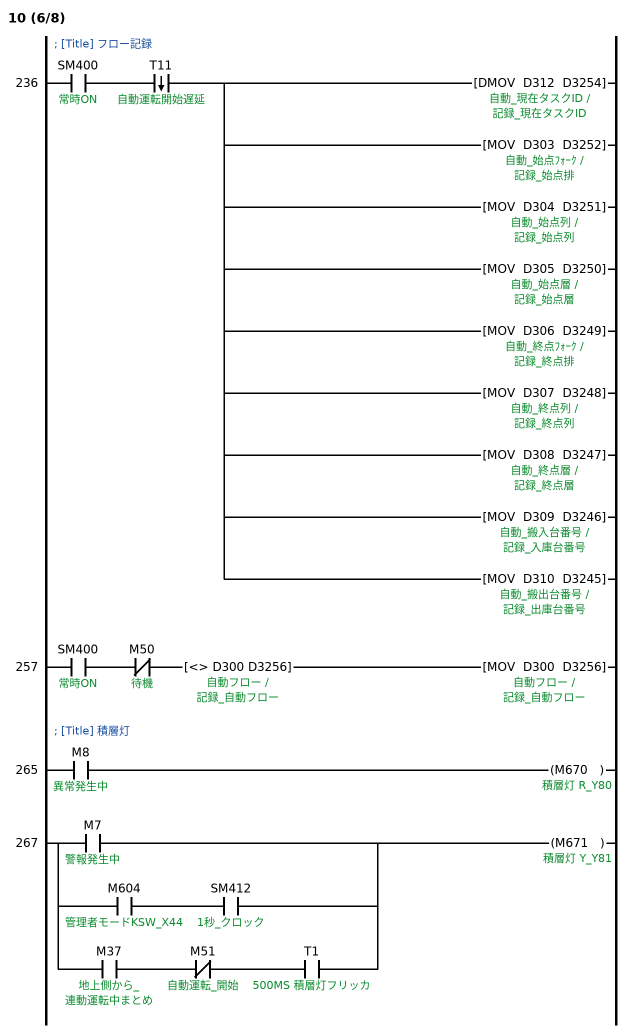
; [Title] フロー記録
236   LD      SM400  ; 常時ON
      ANDF    T11  ; 自動運転開始遅延
      DMOV    D312 D3254  ; 自動_現在タスクID / 記録_現在タスクID
      MOV     D303 D3252  ; 記録_始点排
      MOV     D304 D3251  ; 記録_始点列
      MOV     D305 D3250  ; 記録_始点層
      MOV     D306 D3249  ; 記録_終点排
      MOV     D307 D3248  ; 記録_終点列
      MOV     D308 D3247  ; 記録_終点層
      MOV     D309 D3246  ; 記録_入庫台番号
      MOV     D310 D3245  ; 記録_出庫台番号
257   LD      SM400  ; 常時ON
      ANI     M50  ; 待機
      AND<>   D300 D3256  ; 自動フロー / 記録_自動フロー
      MOV     D300 D3256
; [Title] 積層灯
265   LD      M8  ; 異常発生中
      OUT     M670  ; 積層灯 R_Y80
267   LD      M7  ; 警報発生中
      LD      M604  ; 管理者モードKSW_X44
      AND     SM412  ; 1秒_クロック
      ORB
      LD      M37  ; 地上側から_連動運転中まとめ
      ANI     M51  ; 自動運転_開始
      AND     T1  ; 500MS 積層灯フリッカ
      ORB
      OUT     M671  ; 積層灯 Y_Y81
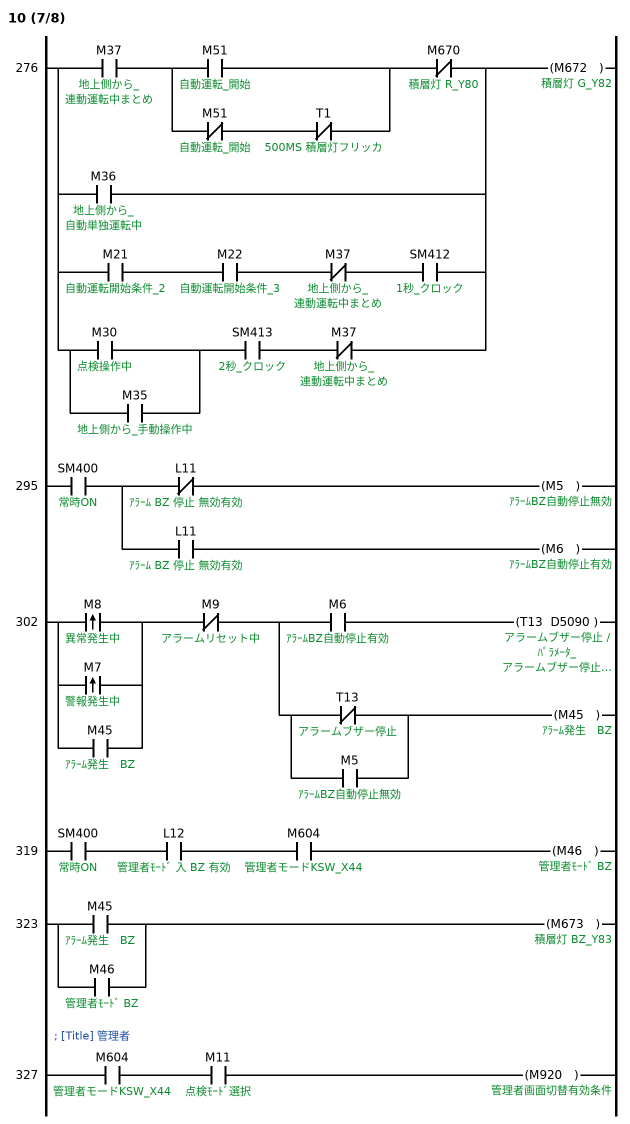
276   LD      M37  ; 地上側から_連動運転中まとめ
      LD      M51  ; 自動運転_開始
      LDI     M51  ; 自動運転_開始
      ANI     T1  ; 500MS 積層灯フリッカ
      ORB
      ANB
      ANI     M670  ; 積層灯 R_Y80
      OR      M36  ; 地上側から_自動単独運転中
      LD      M21  ; 自動運転開始条件_2
      AND     M22  ; 自動運転開始条件_3
      ANI     M37  ; 地上側から_連動運転中まとめ
      AND     SM412  ; 1秒_クロック
      ORB
      LD      M30  ; 点検操作中
      OR      M35  ; 地上側から_手動操作中
      AND     SM413  ; 2秒_クロック
      ANI     M37  ; 地上側から_連動運転中まとめ
      ORB
      OUT     M672  ; 積層灯 G_Y82
295   LD      SM400  ; 常時ON
      MPS
      ANI     L11  ; ｱﾗｰﾑ BZ 停止 無効有効
      OUT     M5  ; ｱﾗｰﾑBZ自動停止無効
      MPP
      AND     L11  ; ｱﾗｰﾑ BZ 停止 無効有効
      OUT     M6  ; ｱﾗｰﾑBZ自動停止有効
302   LDP     M8  ; 異常発生中
      ORP     M7  ; 警報発生中
      OR      M45  ; ｱﾗｰﾑ発生　BZ
      ANI     M9  ; アラームリセット中
      MPS
      AND     M6  ; ｱﾗｰﾑBZ自動停止有効
      OUT     T13 D5090  ; アラームブザー停止 / ﾊﾟﾗﾒｰﾀ_アラームブザー停止設定値
      MPP
      LDI     T13  ; アラームブザー停止
      OR      M5  ; ｱﾗｰﾑBZ自動停止無効
      ANB
      OUT     M45  ; ｱﾗｰﾑ発生　BZ
319   LD      SM400  ; 常時ON
      AND     L12  ; 管理者ﾓｰﾄﾞ 入 BZ 有効
      AND     M604  ; 管理者モードKSW_X44
      OUT     M46  ; 管理者ﾓｰﾄﾞ BZ
323   LD      M45  ; ｱﾗｰﾑ発生　BZ
      OR      M46  ; 管理者ﾓｰﾄﾞ BZ
      OUT     M673  ; 積層灯 BZ_Y83
; [Title] 管理者
327   LD      M604  ; 管理者モードKSW_X44
      AND     M11  ; 点検ﾓｰﾄﾞ選択
      OUT     M920  ; 管理者画面切替有効条件
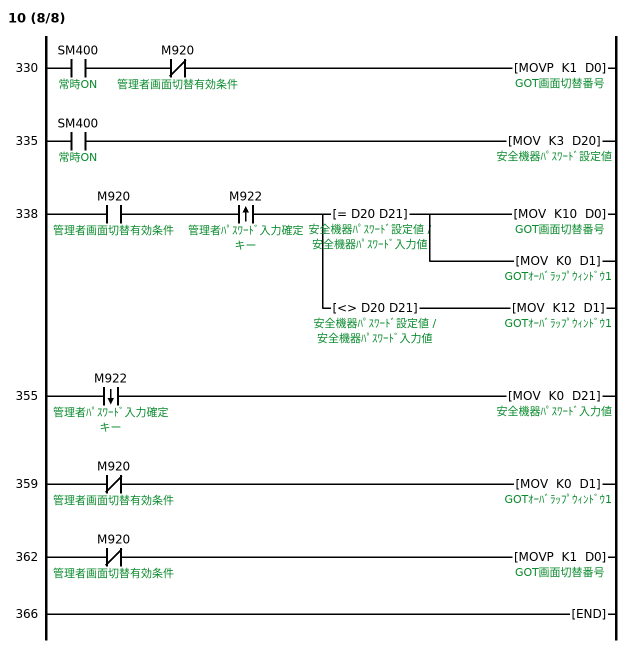
330   LD      SM400  ; 常時ON
      ANI     M920  ; 管理者画面切替有効条件
      MOVP    K1 D0  ; GOT画面切替番号
335   LD      SM400  ; 常時ON
      MOV     K3 D20  ; 安全機器ﾊﾟｽﾜｰﾄﾞ設定値
338   LD      M920  ; 管理者画面切替有効条件
      ANDP    M922  ; 管理者ﾊﾟｽﾜｰﾄﾞ入力確定キー
      MPS
      AND=    D20 D21  ; 安全機器ﾊﾟｽﾜｰﾄﾞ設定値 / 安全機器ﾊﾟｽﾜｰﾄﾞ入力値
      MOV     K10 D0
      MOV     K0 D1  ; GOTｵｰﾊﾞﾗｯﾌﾟｳｨﾝﾄﾞｳ1
      MPP
      AND<>   D20 D21  ; 安全機器ﾊﾟｽﾜｰﾄﾞ設定値 / 安全機器ﾊﾟｽﾜｰﾄﾞ入力値
      MOV     K12 D1
355   LDF     M922  ; 管理者ﾊﾟｽﾜｰﾄﾞ入力確定キー
      MOV     K0 D21
359   LDI     M920  ; 管理者画面切替有効条件
      MOV     K0 D1
362   LDI     M920  ; 管理者画面切替有効条件
      MOVP    K1 D0
366   END
END_PROGRAM

PROGRAM 12  // Stacker制御_自動
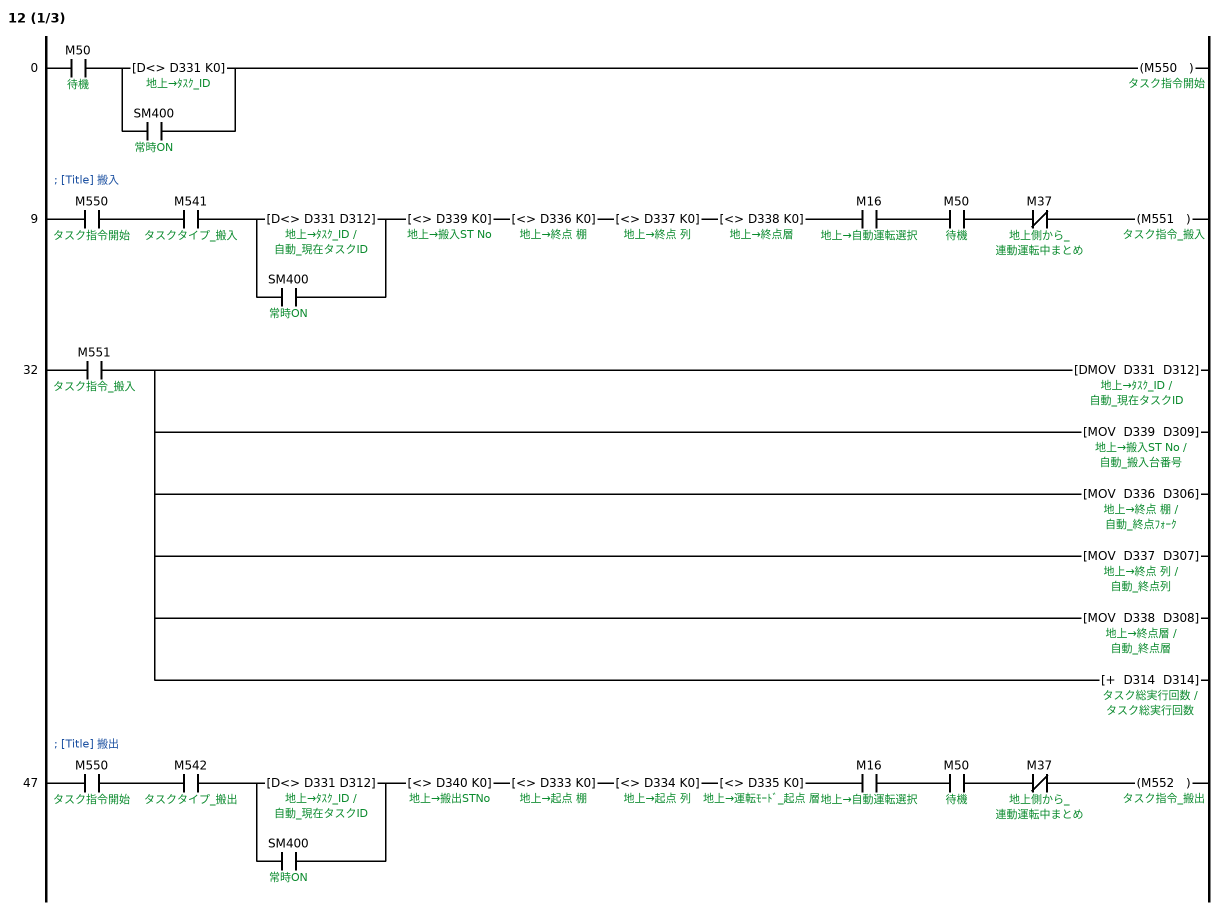
0     LD      M50  ; 待機
      LDD<>   D331 K0  ; 地上→ﾀｽｸ_ID
      OR      SM400  ; 常時ON
      ANB
      OUT     M550  ; タスク指令開始
; [Title] 搬入
9     LD      M550  ; タスク指令開始
      AND     M541  ; タスクタイプ_搬入
      LDD<>   D331 D312  ; 地上→ﾀｽｸ_ID / 自動_現在タスクID
      OR      SM400  ; 常時ON
      ANB
      AND<>   D339 K0  ; 地上→搬入ST No
      AND<>   D336 K0  ; 地上→終点 棚
      AND<>   D337 K0  ; 地上→終点 列
      AND<>   D338 K0  ; 地上→終点層
      AND     M16  ; 地上→自動運転選択
      AND     M50  ; 待機
      ANI     M37  ; 地上側から_連動運転中まとめ
      OUT     M551  ; タスク指令_搬入
32    LD      M551  ; タスク指令_搬入
      DMOV    D331 D312
      MOV     D339 D309  ; 自動_搬入台番号
      MOV     D336 D306  ; 自動_終点ﾌｫｰｸ
      MOV     D337 D307  ; 自動_終点列
      MOV     D338 D308  ; 自動_終点層
      +       D314 D314  ; タスク総実行回数
; [Title] 搬出
47    LD      M550  ; タスク指令開始
      AND     M542  ; タスクタイプ_搬出
      LDD<>   D331 D312  ; 地上→ﾀｽｸ_ID / 自動_現在タスクID
      OR      SM400  ; 常時ON
      ANB
      AND<>   D340 K0  ; 地上→搬出STNo
      AND<>   D333 K0  ; 地上→起点 棚
      AND<>   D334 K0  ; 地上→起点 列
      AND<>   D335 K0  ; 地上→運転ﾓｰﾄﾞ_起点 層
      AND     M16  ; 地上→自動運転選択
      AND     M50  ; 待機
      ANI     M37  ; 地上側から_連動運転中まとめ
      OUT     M552  ; タスク指令_搬出
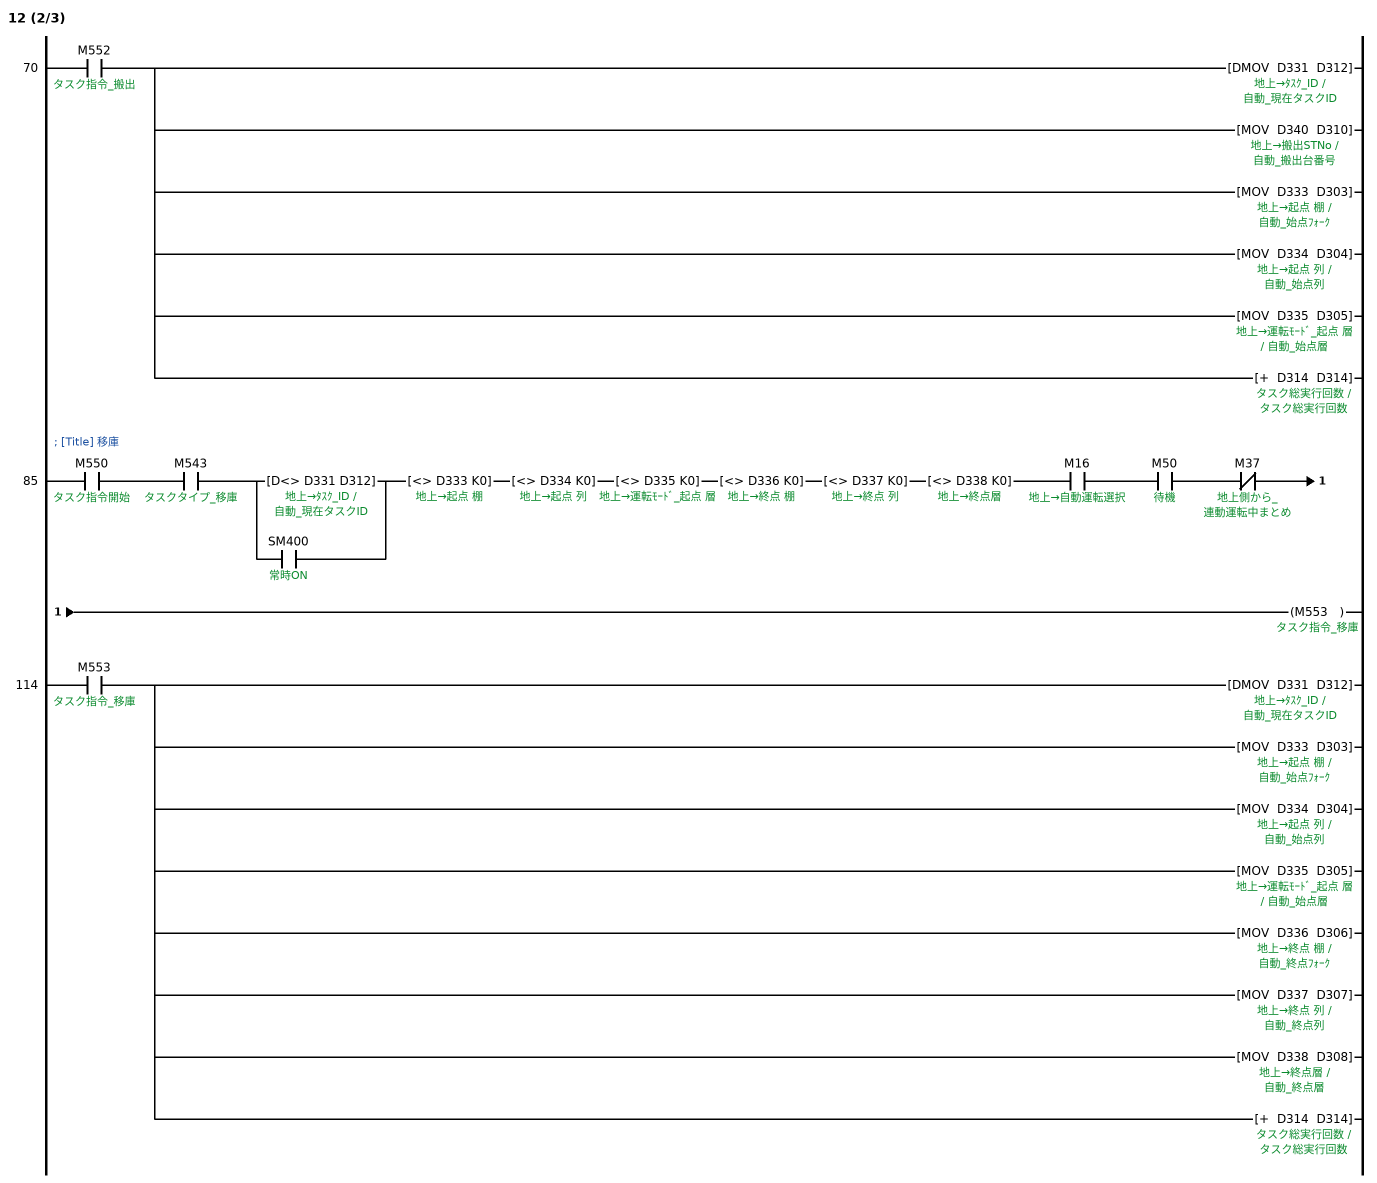
70    LD      M552  ; タスク指令_搬出
      DMOV    D331 D312
      MOV     D340 D310  ; 自動_搬出台番号
      MOV     D333 D303  ; 自動_始点ﾌｫｰｸ
      MOV     D334 D304  ; 自動_始点列
      MOV     D335 D305  ; 自動_始点層
      +       D314 D314
; [Title] 移庫
85    LD      M550  ; タスク指令開始
      AND     M543  ; タスクタイプ_移庫
      LDD<>   D331 D312  ; 地上→ﾀｽｸ_ID / 自動_現在タスクID
      OR      SM400  ; 常時ON
      ANB
      AND<>   D333 K0  ; 地上→起点 棚
      AND<>   D334 K0  ; 地上→起点 列
      AND<>   D335 K0  ; 地上→運転ﾓｰﾄﾞ_起点 層
      AND<>   D336 K0  ; 地上→終点 棚
      AND<>   D337 K0  ; 地上→終点 列
      AND<>   D338 K0  ; 地上→終点層
      AND     M16  ; 地上→自動運転選択
      AND     M50  ; 待機
      ANI     M37  ; 地上側から_連動運転中まとめ
      OUT     M553  ; タスク指令_移庫
114   LD      M553  ; タスク指令_移庫
      DMOV    D331 D312
      MOV     D333 D303
      MOV     D334 D304
      MOV     D335 D305
      MOV     D336 D306
      MOV     D337 D307
      MOV     D338 D308
      +       D314 D314
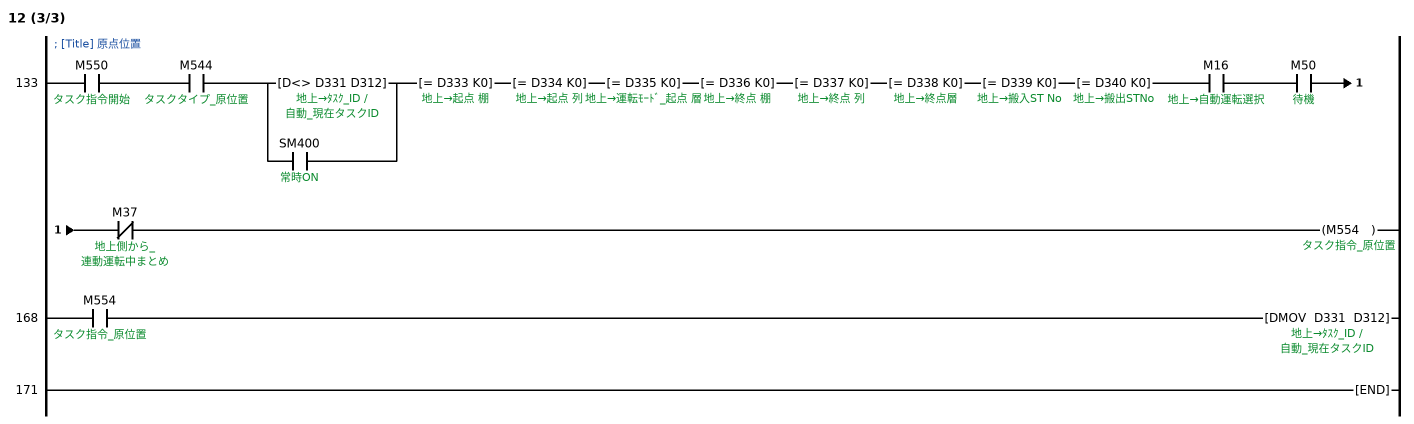
; [Title] 原点位置
133   LD      M550  ; タスク指令開始
      AND     M544  ; タスクタイプ_原位置
      LDD<>   D331 D312  ; 地上→ﾀｽｸ_ID / 自動_現在タスクID
      OR      SM400  ; 常時ON
      ANB
      AND=    D333 K0  ; 地上→起点 棚
      AND=    D334 K0  ; 地上→起点 列
      AND=    D335 K0  ; 地上→運転ﾓｰﾄﾞ_起点 層
      AND=    D336 K0  ; 地上→終点 棚
      AND=    D337 K0  ; 地上→終点 列
      AND=    D338 K0  ; 地上→終点層
      AND=    D339 K0  ; 地上→搬入ST No
      AND=    D340 K0  ; 地上→搬出STNo
      AND     M16  ; 地上→自動運転選択
      AND     M50  ; 待機
      ANI     M37  ; 地上側から_連動運転中まとめ
      OUT     M554  ; タスク指令_原位置
168   LD      M554  ; タスク指令_原位置
      DMOV    D331 D312
171   END
END_PROGRAM

PROGRAM 14  // 点検操作/地上側手動・自動単独
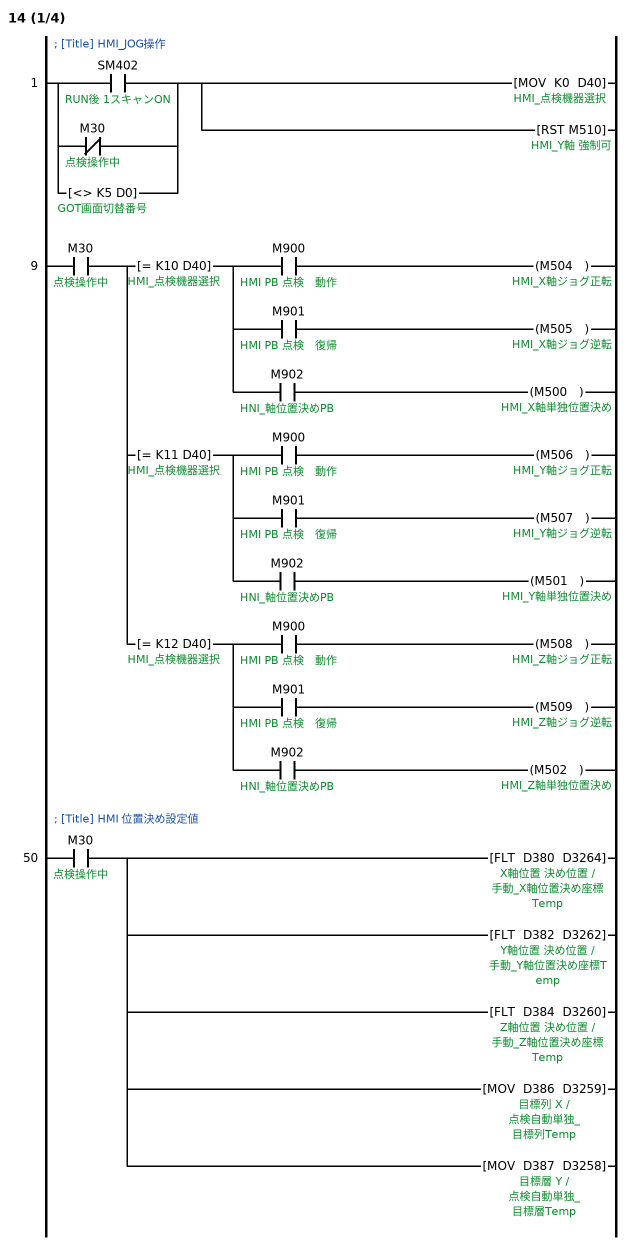
; [Title] HMI_JOG操作
1     LD      SM402  ; RUN後 1スキャンON
      ORI     M30  ; 点検操作中
      OR<>    K5 D0  ; GOT画面切替番号
      MOV     K0 D40  ; HMI_点検機器選択
      RST     M510  ; HMI_Y軸 強制可
9     LD      M30  ; 点検操作中
      MPS
      AND=    K10 D40  ; HMI_点検機器選択
      MPS
      AND     M900  ; HMI PB 点検　動作
      OUT     M504  ; HMI_X軸ジョグ正転
      MRD
      AND     M901  ; HMI PB 点検　復帰
      OUT     M505  ; HMI_X軸ジョグ逆転
      MPP
      AND     M902  ; HNI_軸位置決めPB
      OUT     M500  ; HMI_X軸単独位置決め
      MRD
      AND=    K11 D40  ; HMI_点検機器選択
      MPS
      AND     M900  ; HMI PB 点検　動作
      OUT     M506  ; HMI_Y軸ジョグ正転
      MRD
      AND     M901  ; HMI PB 点検　復帰
      OUT     M507  ; HMI_Y軸ジョグ逆転
      MPP
      AND     M902  ; HNI_軸位置決めPB
      OUT     M501  ; HMI_Y軸単独位置決め
      MPP
      AND=    K12 D40  ; HMI_点検機器選択
      MPS
      AND     M900  ; HMI PB 点検　動作
      OUT     M508  ; HMI_Z軸ジョグ正転
      MRD
      AND     M901  ; HMI PB 点検　復帰
      OUT     M509  ; HMI_Z軸ジョグ逆転
      MPP
      AND     M902  ; HNI_軸位置決めPB
      OUT     M502  ; HMI_Z軸単独位置決め
; [Title] HMI 位置決め設定値
50    LD      M30  ; 点検操作中
      FLT     D380 D3264  ; X軸位置 決め位置 / 手動_X軸位置決め座標Temp
      FLT     D382 D3262  ; Y軸位置 決め位置 / 手動_Y軸位置決め座標Temp
      FLT     D384 D3260  ; Z軸位置 決め位置 / 手動_Z軸位置決め座標Temp
      MOV     D386 D3259  ; 目標列 X / 点検自動単独_目標列Temp
      MOV     D387 D3258  ; 目標層 Y / 点検自動単独_目標層Temp
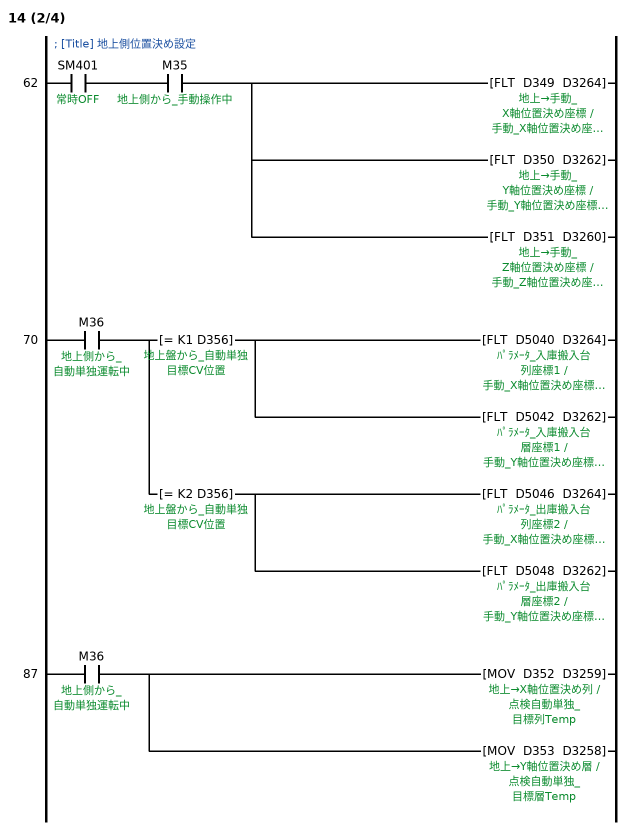
; [Title] 地上側位置決め設定
62    LD      SM401  ; 常時OFF
      AND     M35  ; 地上側から_手動操作中
      FLT     D349 D3264  ; 地上→手動_X軸位置決め座標
      FLT     D350 D3262  ; 地上→手動_Y軸位置決め座標
      FLT     D351 D3260  ; 地上→手動_Z軸位置決め座標
70    LD      M36  ; 地上側から_自動単独運転中
      MPS
      AND=    K1 D356  ; 地上盤から_自動単独 目標CV位置
      FLT     D5040 D3264  ; ﾊﾟﾗﾒｰﾀ_入庫搬入台  列座標1
      FLT     D5042 D3262  ; ﾊﾟﾗﾒｰﾀ_入庫搬入台  層座標1
      MPP
      AND=    K2 D356  ; 地上盤から_自動単独 目標CV位置
      FLT     D5046 D3264  ; ﾊﾟﾗﾒｰﾀ_出庫搬入台  列座標2
      FLT     D5048 D3262  ; ﾊﾟﾗﾒｰﾀ_出庫搬入台  層座標2
87    LD      M36  ; 地上側から_自動単独運転中
      MOV     D352 D3259  ; 地上→X軸位置決め列
      MOV     D353 D3258  ; 地上→Y軸位置決め層
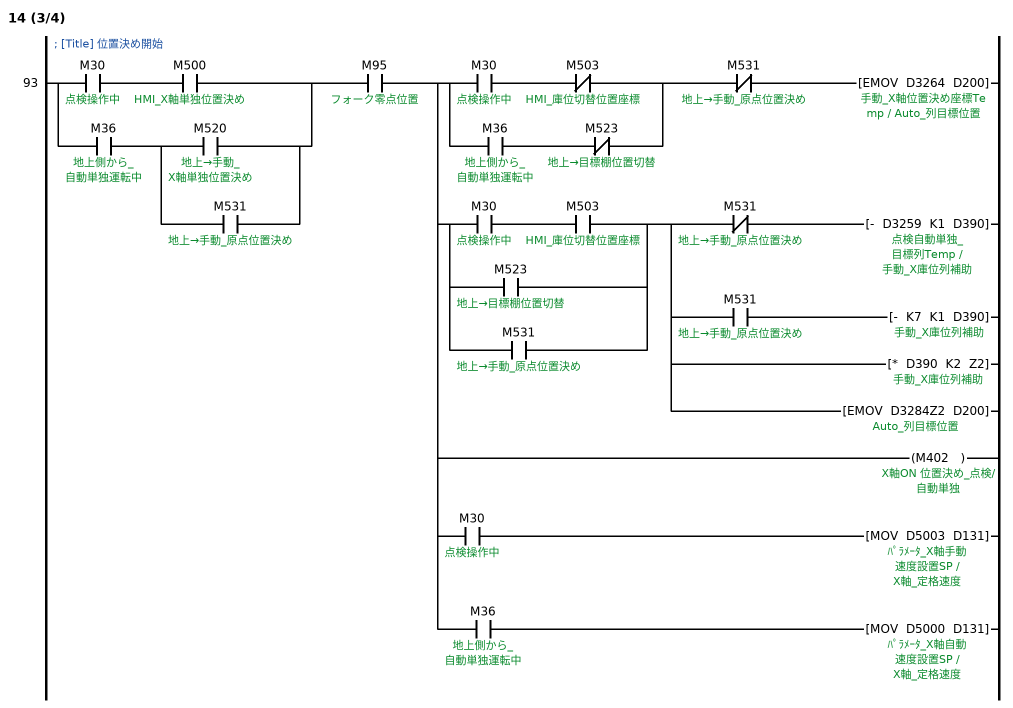
; [Title] 位置決め開始
93    LD      M30  ; 点検操作中
      AND     M500  ; HMI_X軸単独位置決め
      LD      M36  ; 地上側から_自動単独運転中
      LD      M520  ; 地上→手動_X軸単独位置決め
      OR      M531  ; 地上→手動_原点位置決め
      ANB
      ORB
      AND     M95  ; フォーク零点位置
      MPS
      LD      M30  ; 点検操作中
      ANI     M503  ; HMI_庫位切替位置座標
      LD      M36  ; 地上側から_自動単独運転中
      ANI     M523  ; 地上→目標棚位置切替
      ORB
      ANB
      ANI     M531  ; 地上→手動_原点位置決め
      EMOV    D3264 D200  ; Auto_列目標位置
      MRD
      LD      M30  ; 点検操作中
      AND     M503  ; HMI_庫位切替位置座標
      OR      M523  ; 地上→目標棚位置切替
      OR      M531  ; 地上→手動_原点位置決め
      ANB
      MPS
      ANI     M531  ; 地上→手動_原点位置決め
      -       D3259 K1 D390  ; 手動_X庫位列補助
      MRD
      AND     M531  ; 地上→手動_原点位置決め
      -       K7 K1 D390
      MPP
      *       D390 K2 Z2
      EMOV    D3284Z2 D200
      MPP
      OUT     M402  ; X軸ON 位置決め_点検/自動単独
      MPS
      AND     M30  ; 点検操作中
      MOV     D5003 D131  ; ﾊﾟﾗﾒｰﾀ_X軸手動 速度設置SP / X軸_定格速度
      MPP
      AND     M36  ; 地上側から_自動単独運転中
      MOV     D5000 D131  ; ﾊﾟﾗﾒｰﾀ_X軸自動 速度設置SP
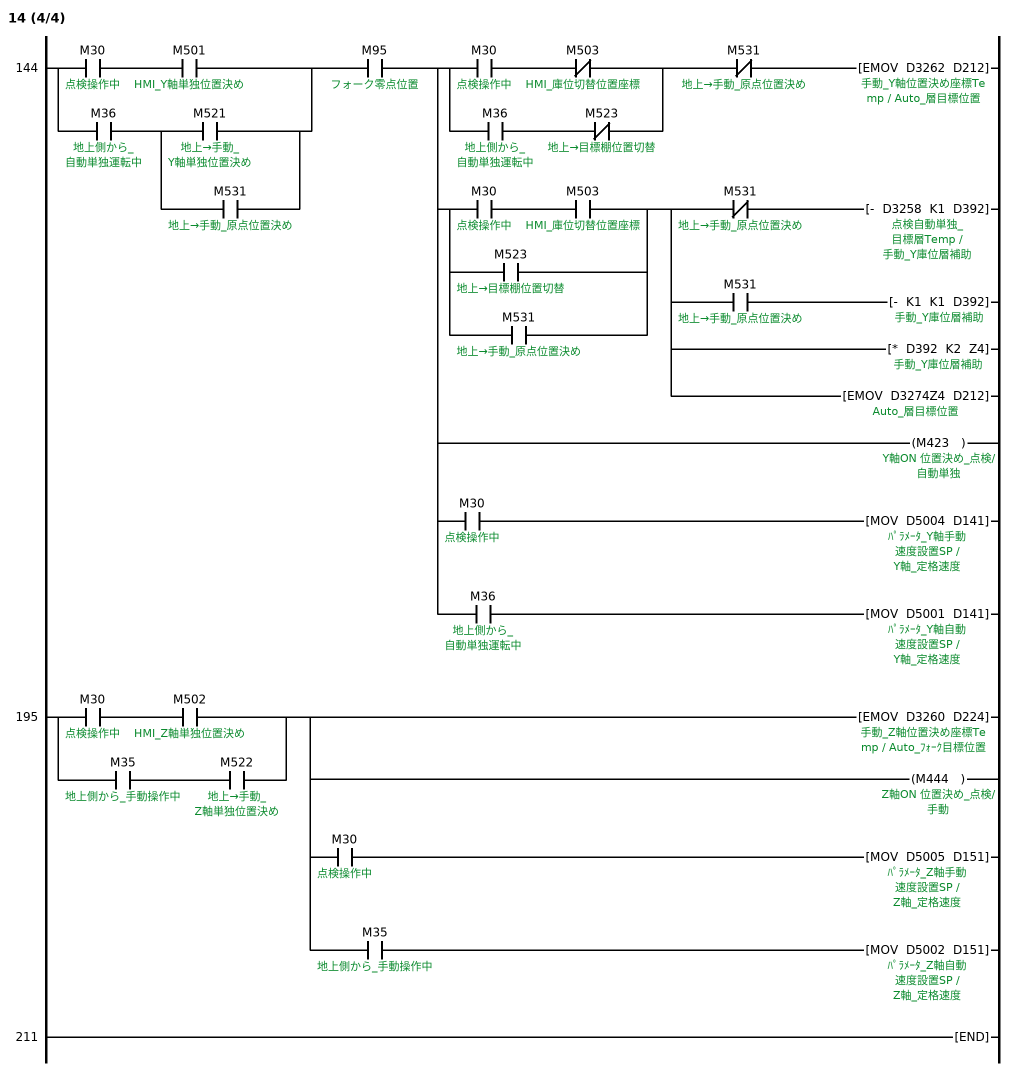
144   LD      M30  ; 点検操作中
      AND     M501  ; HMI_Y軸単独位置決め
      LD      M36  ; 地上側から_自動単独運転中
      LD      M521  ; 地上→手動_Y軸単独位置決め
      OR      M531  ; 地上→手動_原点位置決め
      ANB
      ORB
      AND     M95  ; フォーク零点位置
      MPS
      LD      M30  ; 点検操作中
      ANI     M503  ; HMI_庫位切替位置座標
      LD      M36  ; 地上側から_自動単独運転中
      ANI     M523  ; 地上→目標棚位置切替
      ORB
      ANB
      ANI     M531  ; 地上→手動_原点位置決め
      EMOV    D3262 D212  ; Auto_層目標位置
      MRD
      LD      M30  ; 点検操作中
      AND     M503  ; HMI_庫位切替位置座標
      OR      M523  ; 地上→目標棚位置切替
      OR      M531  ; 地上→手動_原点位置決め
      ANB
      MPS
      ANI     M531  ; 地上→手動_原点位置決め
      -       D3258 K1 D392  ; 手動_Y庫位層補助
      MRD
      AND     M531  ; 地上→手動_原点位置決め
      -       K1 K1 D392
      MPP
      *       D392 K2 Z4
      EMOV    D3274Z4 D212
      MPP
      OUT     M423  ; Y軸ON 位置決め_点検/自動単独
      MPS
      AND     M30  ; 点検操作中
      MOV     D5004 D141  ; ﾊﾟﾗﾒｰﾀ_Y軸手動 速度設置SP / Y軸_定格速度
      MPP
      AND     M36  ; 地上側から_自動単独運転中
      MOV     D5001 D141  ; ﾊﾟﾗﾒｰﾀ_Y軸自動 速度設置SP
195   LD      M30  ; 点検操作中
      AND     M502  ; HMI_Z軸単独位置決め
      LD      M35  ; 地上側から_手動操作中
      AND     M522  ; 地上→手動_Z軸単独位置決め
      ORB
      EMOV    D3260 D224  ; Auto_ﾌｫｰｸ目標位置
      OUT     M444  ; Z軸ON 位置決め_点検/手動
      MPS
      AND     M30  ; 点検操作中
      MOV     D5005 D151  ; ﾊﾟﾗﾒｰﾀ_Z軸手動 速度設置SP / Z軸_定格速度
      MPP
      AND     M35  ; 地上側から_手動操作中
      MOV     D5002 D151  ; ﾊﾟﾗﾒｰﾀ_Z軸自動 速度設置SP
211   END
END_PROGRAM

PROGRAM 15  // 軸制御
VAR
  AO1 : INT;
  __IST_24fe211bdc5e490f : I+ST_24fe211bdc5e490f;
  __IST_2ed1eb90aebe4c54 : I+ST_2ed1eb90aebe4c54;
  AO2 : INT;
END_VAR
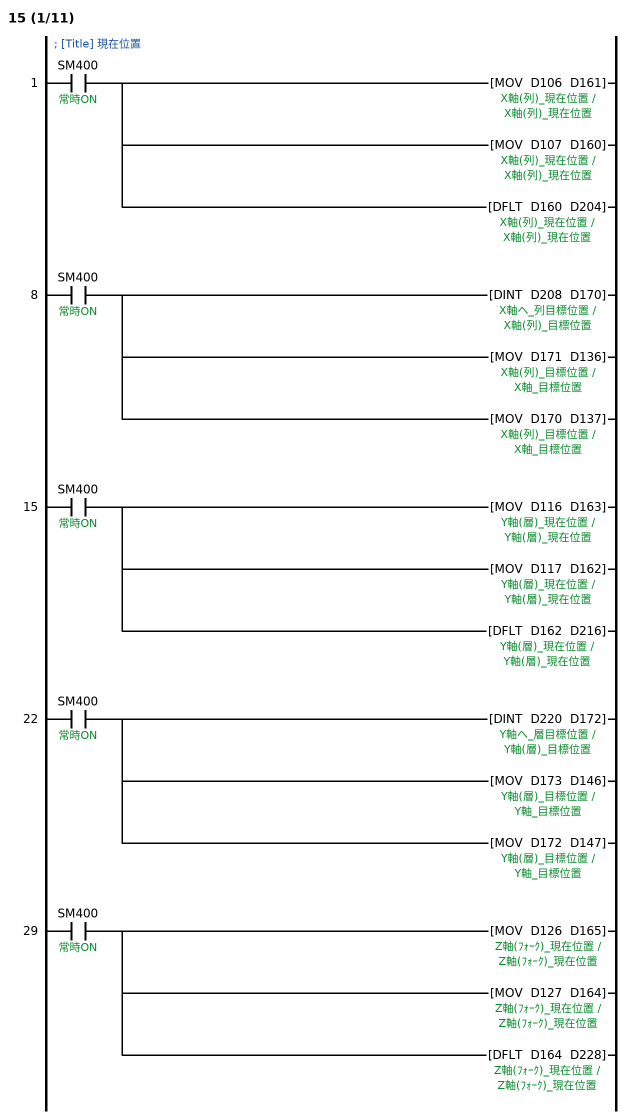
; [Title] 現在位置
1     LD      SM400  ; 常時ON
      MOV     D106 D161  ; X軸(列)_現在位置 / X軸(列)_現在位置
      MOV     D107 D160  ; X軸(列)_現在位置 / X軸(列)_現在位置
      DFLT    D160 D204  ; X軸(列)_現在位置
8     LD      SM400  ; 常時ON
      DINT    D208 D170  ; X軸へ_列目標位置 / X軸(列)_目標位置
      MOV     D171 D136  ; X軸(列)_目標位置 / X軸_目標位置
      MOV     D170 D137  ; X軸_目標位置
15    LD      SM400  ; 常時ON
      MOV     D116 D163  ; Y軸(層)_現在位置 / Y軸(層)_現在位置
      MOV     D117 D162  ; Y軸(層)_現在位置 / Y軸(層)_現在位置
      DFLT    D162 D216  ; Y軸(層)_現在位置
22    LD      SM400  ; 常時ON
      DINT    D220 D172  ; Y軸へ_層目標位置 / Y軸(層)_目標位置
      MOV     D173 D146  ; Y軸(層)_目標位置 / Y軸_目標位置
      MOV     D172 D147  ; Y軸_目標位置
29    LD      SM400  ; 常時ON
      MOV     D126 D165  ; Z軸(ﾌｫｰｸ)_現在位置 / Z軸(ﾌｫｰｸ)_現在位置
      MOV     D127 D164  ; Z軸(ﾌｫｰｸ)_現在位置 / Z軸(ﾌｫｰｸ)_現在位置
      DFLT    D164 D228  ; Z軸(ﾌｫｰｸ)_現在位置
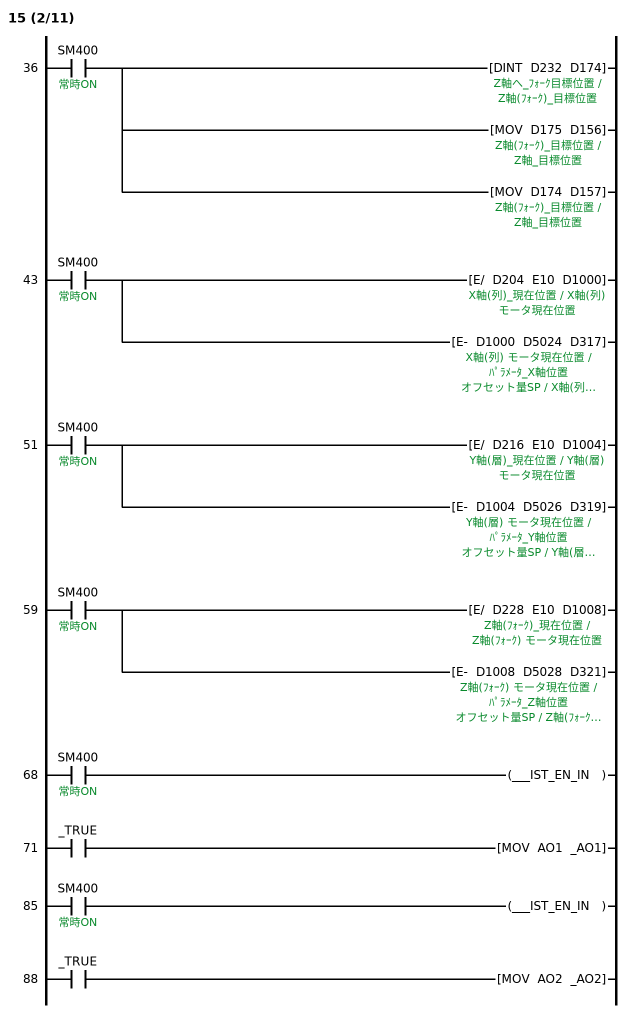
36    LD      SM400  ; 常時ON
      DINT    D232 D174  ; Z軸へ_ﾌｫｰｸ目標位置 / Z軸(ﾌｫｰｸ)_目標位置
      MOV     D175 D156  ; Z軸(ﾌｫｰｸ)_目標位置 / Z軸_目標位置
      MOV     D174 D157  ; Z軸_目標位置
43    LD      SM400  ; 常時ON
      E/      D204 E10 D1000  ; X軸(列) モータ現在位置
      E-      D1000 D5024 D317  ; ﾊﾟﾗﾒｰﾀ_X軸位置 オフセット量SP / X軸(列) 現在位置
51    LD      SM400  ; 常時ON
      E/      D216 E10 D1004  ; Y軸(層) モータ現在位置
      E-      D1004 D5026 D319  ; ﾊﾟﾗﾒｰﾀ_Y軸位置 オフセット量SP / Y軸(層) 現在位置
59    LD      SM400  ; 常時ON
      E/      D228 E10 D1008  ; Z軸(ﾌｫｰｸ) モータ現在位置
      E-      D1008 D5028 D321  ; ﾊﾟﾗﾒｰﾀ_Z軸位置 オフセット量SP / Z軸(ﾌｫｰｸ) 現在位置
; FB BLK START I+ST_24fe211bdc5e490f(__IST_24fe211bdc5e490f)
68    LD      SM400  ; 常時ON
      OUT     ___IST_EN_IN
71    LD      _TRUE
      MOV     AO1 _AO1
; FB START
; FB_NAME I+ST_24fe211bdc5e490f
; INSTANCE_NAME __IST_24fe211bdc5e490f
; FB IN_B:__IST_EN_IN
; FB OUT___IST_EN_OUT:B
; FB IN_W:AO1
; FB OUT_AO1:W
; FB END
; FB BLK END
; FB BLK START I+ST_2ed1eb90aebe4c54(__IST_2ed1eb90aebe4c54)
85    LD      SM400  ; 常時ON
      OUT     ___IST_EN_IN
88    LD      _TRUE
      MOV     AO2 _AO2
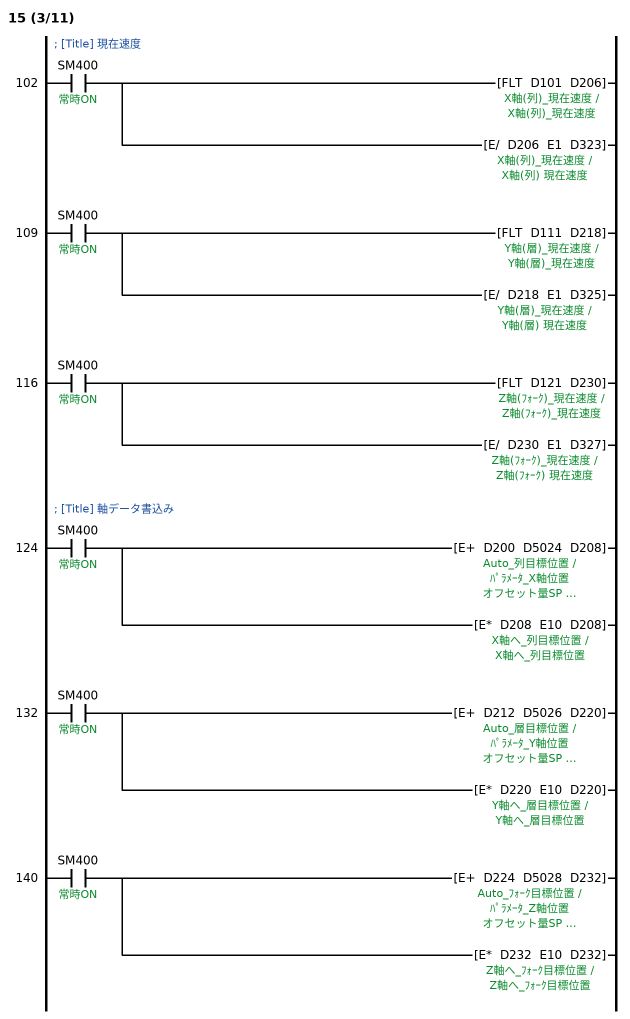
; FB START
; FB_NAME I+ST_2ed1eb90aebe4c54
; INSTANCE_NAME __IST_2ed1eb90aebe4c54
; FB IN_B:__IST_EN_IN
; FB OUT___IST_EN_OUT:B
; FB IN_W:AO2
; FB OUT_AO2:W
; FB END
; FB BLK END
; [Title] 現在速度
102   LD      SM400  ; 常時ON
      FLT     D101 D206  ; X軸(列)_現在速度 / X軸(列)_現在速度
      E/      D206 E1 D323  ; X軸(列) 現在速度
109   LD      SM400  ; 常時ON
      FLT     D111 D218  ; Y軸(層)_現在速度 / Y軸(層)_現在速度
      E/      D218 E1 D325  ; Y軸(層) 現在速度
116   LD      SM400  ; 常時ON
      FLT     D121 D230  ; Z軸(ﾌｫｰｸ)_現在速度 / Z軸(ﾌｫｰｸ)_現在速度
      E/      D230 E1 D327  ; Z軸(ﾌｫｰｸ) 現在速度
; [Title] 軸データ書込み
124   LD      SM400  ; 常時ON
      E+      D200 D5024 D208  ; Auto_列目標位置
      E*      D208 E10 D208
132   LD      SM400  ; 常時ON
      E+      D212 D5026 D220  ; Auto_層目標位置
      E*      D220 E10 D220
140   LD      SM400  ; 常時ON
      E+      D224 D5028 D232  ; Auto_ﾌｫｰｸ目標位置
      E*      D232 E10 D232
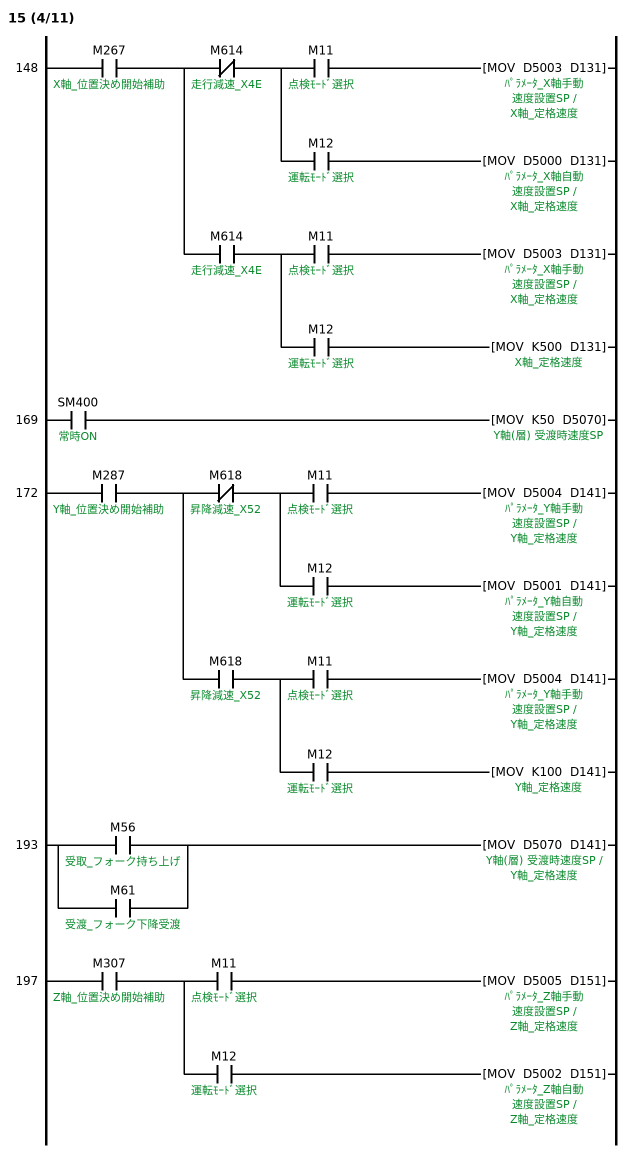
148   LD      M267  ; X軸_位置決め開始補助
      MPS
      ANI     M614  ; 走行減速_X4E
      MPS
      AND     M11  ; 点検ﾓｰﾄﾞ選択
      MOV     D5003 D131  ; ﾊﾟﾗﾒｰﾀ_X軸手動 速度設置SP / X軸_定格速度
      MPP
      AND     M12  ; 運転ﾓｰﾄﾞ選択
      MOV     D5000 D131  ; ﾊﾟﾗﾒｰﾀ_X軸自動 速度設置SP
      MPP
      AND     M614  ; 走行減速_X4E
      MPS
      AND     M11  ; 点検ﾓｰﾄﾞ選択
      MOV     D5003 D131
      MPP
      AND     M12  ; 運転ﾓｰﾄﾞ選択
      MOV     K500 D131
169   LD      SM400  ; 常時ON
      MOV     K50 D5070  ; Y軸(層) 受渡時速度SP
172   LD      M287  ; Y軸_位置決め開始補助
      MPS
      ANI     M618  ; 昇降減速_X52
      MPS
      AND     M11  ; 点検ﾓｰﾄﾞ選択
      MOV     D5004 D141  ; ﾊﾟﾗﾒｰﾀ_Y軸手動 速度設置SP / Y軸_定格速度
      MPP
      AND     M12  ; 運転ﾓｰﾄﾞ選択
      MOV     D5001 D141  ; ﾊﾟﾗﾒｰﾀ_Y軸自動 速度設置SP
      MPP
      AND     M618  ; 昇降減速_X52
      MPS
      AND     M11  ; 点検ﾓｰﾄﾞ選択
      MOV     D5004 D141
      MPP
      AND     M12  ; 運転ﾓｰﾄﾞ選択
      MOV     K100 D141
193   LD      M56  ; 受取_フォーク持ち上げ
      OR      M61  ; 受渡_フォーク下降受渡
      MOV     D5070 D141
197   LD      M307  ; Z軸_位置決め開始補助
      MPS
      AND     M11  ; 点検ﾓｰﾄﾞ選択
      MOV     D5005 D151  ; ﾊﾟﾗﾒｰﾀ_Z軸手動 速度設置SP / Z軸_定格速度
      MPP
      AND     M12  ; 運転ﾓｰﾄﾞ選択
      MOV     D5002 D151  ; ﾊﾟﾗﾒｰﾀ_Z軸自動 速度設置SP
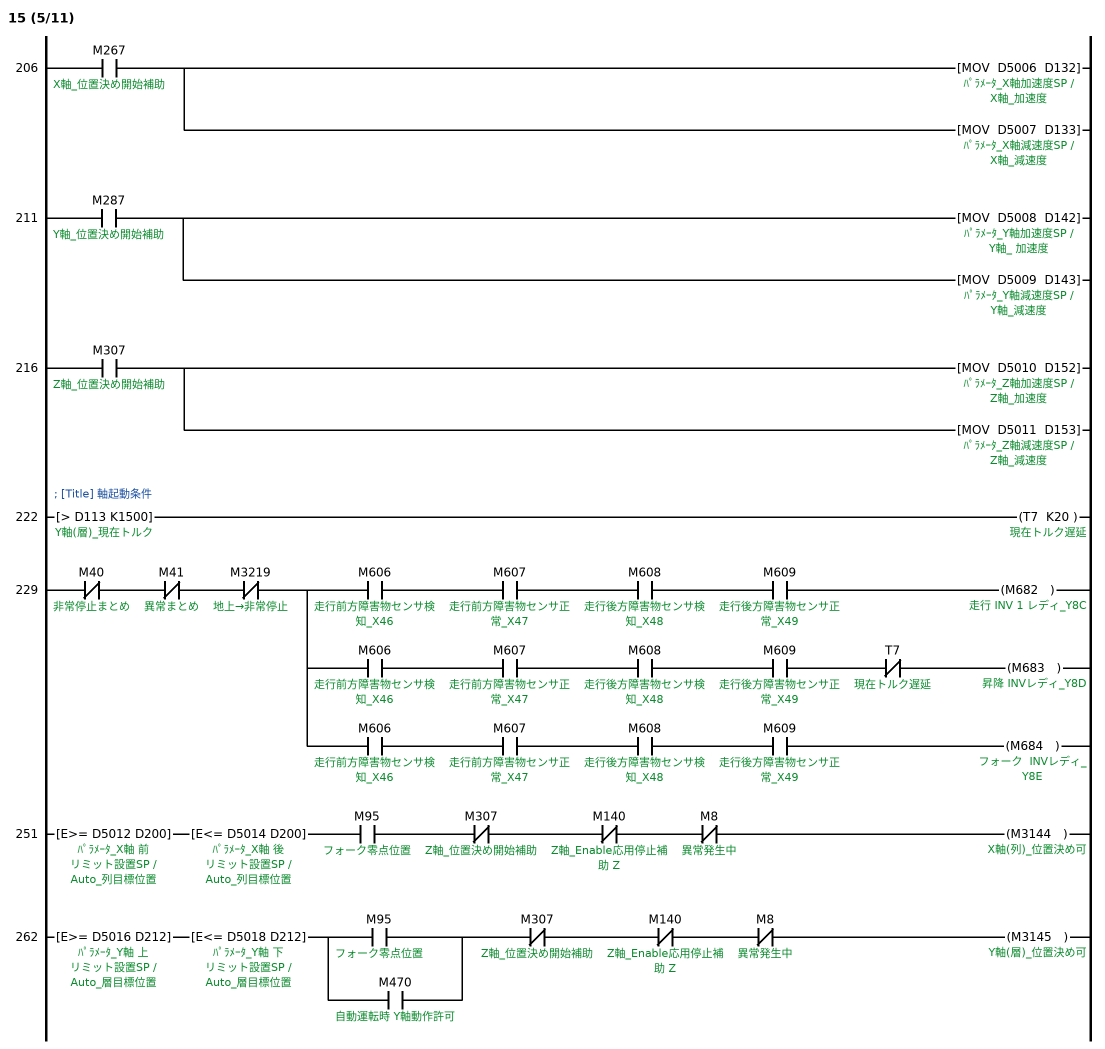
206   LD      M267  ; X軸_位置決め開始補助
      MOV     D5006 D132  ; ﾊﾟﾗﾒｰﾀ_X軸加速度SP / X軸_加速度
      MOV     D5007 D133  ; ﾊﾟﾗﾒｰﾀ_X軸減速度SP / X軸_減速度
211   LD      M287  ; Y軸_位置決め開始補助
      MOV     D5008 D142  ; ﾊﾟﾗﾒｰﾀ_Y軸加速度SP / Y軸_ 加速度
      MOV     D5009 D143  ; ﾊﾟﾗﾒｰﾀ_Y軸減速度SP / Y軸_減速度
216   LD      M307  ; Z軸_位置決め開始補助
      MOV     D5010 D152  ; ﾊﾟﾗﾒｰﾀ_Z軸加速度SP / Z軸_加速度
      MOV     D5011 D153  ; ﾊﾟﾗﾒｰﾀ_Z軸減速度SP / Z軸_減速度
; [Title] 軸起動条件
222   LD>     D113 K1500  ; Y軸(層)_現在トルク
      OUT     T7 K20  ; 現在トルク遅延
229   LDI     M40  ; 非常停止まとめ
      ANI     M41  ; 異常まとめ
      ANI     M3219  ; 地上→非常停止
      MPS
      AND     M606  ; 走行前方障害物センサ検知_X46
      AND     M607  ; 走行前方障害物センサ正常_X47
      AND     M608  ; 走行後方障害物センサ検知_X48
      AND     M609  ; 走行後方障害物センサ正常_X49
      OUT     M682  ; 走行 INV 1 レディ_Y8C
      MRD
      AND     M606  ; 走行前方障害物センサ検知_X46
      AND     M607  ; 走行前方障害物センサ正常_X47
      AND     M608  ; 走行後方障害物センサ検知_X48
      AND     M609  ; 走行後方障害物センサ正常_X49
      ANI     T7  ; 現在トルク遅延
      OUT     M683  ; 昇降 INVレディ_Y8D
      MPP
      AND     M606  ; 走行前方障害物センサ検知_X46
      AND     M607  ; 走行前方障害物センサ正常_X47
      AND     M608  ; 走行後方障害物センサ検知_X48
      AND     M609  ; 走行後方障害物センサ正常_X49
      OUT     M684  ; フォーク  INVレディ_Y8E
251   LDE>=   D5012 D200  ; ﾊﾟﾗﾒｰﾀ_X軸 前 リミット設置SP / Auto_列目標位置
      ANDE<=  D5014 D200  ; ﾊﾟﾗﾒｰﾀ_X軸 後 リミット設置SP / Auto_列目標位置
      AND     M95  ; フォーク零点位置
      ANI     M307  ; Z軸_位置決め開始補助
      ANI     M140  ; Z軸_Enable応用停止補助 Z
      ANI     M8  ; 異常発生中
      OUT     M3144  ; X軸(列)_位置決め可
262   LDE>=   D5016 D212  ; ﾊﾟﾗﾒｰﾀ_Y軸 上 リミット設置SP / Auto_層目標位置
      ANDE<=  D5018 D212  ; ﾊﾟﾗﾒｰﾀ_Y軸 下 リミット設置SP / Auto_層目標位置
      LD      M95  ; フォーク零点位置
      OR      M470  ; 自動運転時 Y軸動作許可
      ANB
      ANI     M307  ; Z軸_位置決め開始補助
      ANI     M140  ; Z軸_Enable応用停止補助 Z
      ANI     M8  ; 異常発生中
      OUT     M3145  ; Y軸(層)_位置決め可
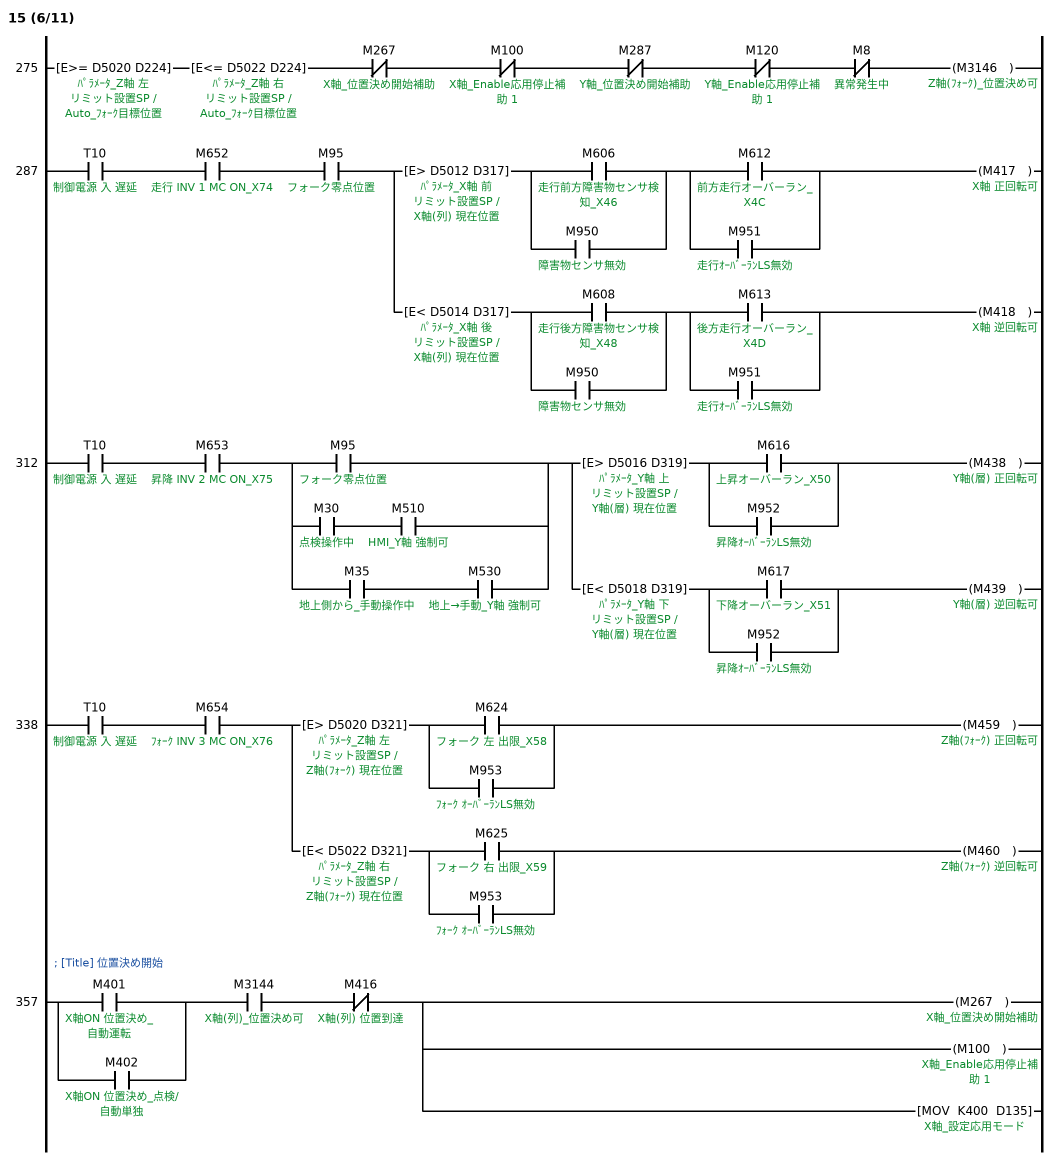
275   LDE>=   D5020 D224  ; ﾊﾟﾗﾒｰﾀ_Z軸 左 リミット設置SP / Auto_ﾌｫｰｸ目標位置
      ANDE<=  D5022 D224  ; ﾊﾟﾗﾒｰﾀ_Z軸 右 リミット設置SP / Auto_ﾌｫｰｸ目標位置
      ANI     M267  ; X軸_位置決め開始補助
      ANI     M100  ; X軸_Enable応用停止補助 1
      ANI     M287  ; Y軸_位置決め開始補助
      ANI     M120  ; Y軸_Enable応用停止補助 1
      ANI     M8  ; 異常発生中
      OUT     M3146  ; Z軸(ﾌｫｰｸ)_位置決め可
287   LD      T10  ; 制御電源 入 遅延
      AND     M652  ; 走行 INV 1 MC ON_X74
      AND     M95  ; フォーク零点位置
      MPS
      ANDE>   D5012 D317  ; ﾊﾟﾗﾒｰﾀ_X軸 前 リミット設置SP / X軸(列) 現在位置
      LD      M606  ; 走行前方障害物センサ検知_X46
      OR      M950  ; 障害物センサ無効
      ANB
      LD      M612  ; 前方走行オーバーラン_X4C
      OR      M951  ; 走行ｵｰﾊﾞｰﾗﾝLS無効
      ANB
      OUT     M417  ; X軸 正回転可
      MPP
      ANDE<   D5014 D317  ; ﾊﾟﾗﾒｰﾀ_X軸 後 リミット設置SP / X軸(列) 現在位置
      LD      M608  ; 走行後方障害物センサ検知_X48
      OR      M950  ; 障害物センサ無効
      ANB
      LD      M613  ; 後方走行オーバーラン_X4D
      OR      M951  ; 走行ｵｰﾊﾞｰﾗﾝLS無効
      ANB
      OUT     M418  ; X軸 逆回転可
312   LD      T10  ; 制御電源 入 遅延
      AND     M653  ; 昇降 INV 2 MC ON_X75
      LD      M95  ; フォーク零点位置
      LD      M30  ; 点検操作中
      AND     M510  ; HMI_Y軸 強制可
      ORB
      LD      M35  ; 地上側から_手動操作中
      AND     M530  ; 地上→手動_Y軸 強制可
      ORB
      ANB
      MPS
      ANDE>   D5016 D319  ; ﾊﾟﾗﾒｰﾀ_Y軸 上 リミット設置SP / Y軸(層) 現在位置
      LD      M616  ; 上昇オーバーラン_X50
      OR      M952  ; 昇降ｵｰﾊﾞｰﾗﾝLS無効
      ANB
      OUT     M438  ; Y軸(層) 正回転可
      MPP
      ANDE<   D5018 D319  ; ﾊﾟﾗﾒｰﾀ_Y軸 下 リミット設置SP / Y軸(層) 現在位置
      LD      M617  ; 下降オーバーラン_X51
      OR      M952  ; 昇降ｵｰﾊﾞｰﾗﾝLS無効
      ANB
      OUT     M439  ; Y軸(層) 逆回転可
338   LD      T10  ; 制御電源 入 遅延
      AND     M654  ; ﾌｫｰｸ INV 3 MC ON_X76
      MPS
      ANDE>   D5020 D321  ; ﾊﾟﾗﾒｰﾀ_Z軸 左 リミット設置SP / Z軸(ﾌｫｰｸ) 現在位置
      LD      M624  ; フォーク 左 出限_X58
      OR      M953  ; ﾌｫｰｸ ｵｰﾊﾞｰﾗﾝLS無効
      ANB
      OUT     M459  ; Z軸(ﾌｫｰｸ) 正回転可
      MPP
      ANDE<   D5022 D321  ; ﾊﾟﾗﾒｰﾀ_Z軸 右 リミット設置SP / Z軸(ﾌｫｰｸ) 現在位置
      LD      M625  ; フォーク 右 出限_X59
      OR      M953  ; ﾌｫｰｸ ｵｰﾊﾞｰﾗﾝLS無効
      ANB
      OUT     M460  ; Z軸(ﾌｫｰｸ) 逆回転可
; [Title] 位置決め開始
357   LD      M401  ; X軸ON 位置決め_自動運転
      OR      M402  ; X軸ON 位置決め_点検/自動単独
      AND     M3144  ; X軸(列)_位置決め可
      ANI     M416  ; X軸(列) 位置到達
      OUT     M267  ; X軸_位置決め開始補助
      OUT     M100  ; X軸_Enable応用停止補助 1
      MOV     K400 D135  ; X軸_設定応用モード
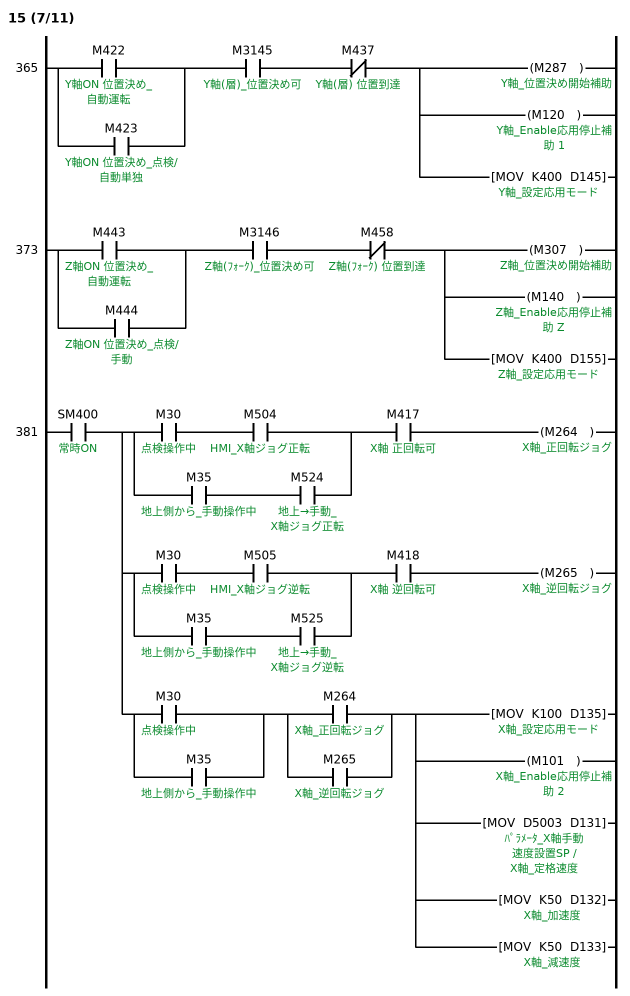
365   LD      M422  ; Y軸ON 位置決め_自動運転
      OR      M423  ; Y軸ON 位置決め_点検/自動単独
      AND     M3145  ; Y軸(層)_位置決め可
      ANI     M437  ; Y軸(層) 位置到達
      OUT     M287  ; Y軸_位置決め開始補助
      OUT     M120  ; Y軸_Enable応用停止補助 1
      MOV     K400 D145  ; Y軸_設定応用モード
373   LD      M443  ; Z軸ON 位置決め_自動運転
      OR      M444  ; Z軸ON 位置決め_点検/手動
      AND     M3146  ; Z軸(ﾌｫｰｸ)_位置決め可
      ANI     M458  ; Z軸(ﾌｫｰｸ) 位置到達
      OUT     M307  ; Z軸_位置決め開始補助
      OUT     M140  ; Z軸_Enable応用停止補助 Z
      MOV     K400 D155  ; Z軸_設定応用モード
381   LD      SM400  ; 常時ON
      MPS
      LD      M30  ; 点検操作中
      AND     M504  ; HMI_X軸ジョグ正転
      LD      M35  ; 地上側から_手動操作中
      AND     M524  ; 地上→手動_X軸ジョグ正転
      ORB
      ANB
      AND     M417  ; X軸 正回転可
      OUT     M264  ; X軸_正回転ジョグ
      MRD
      LD      M30  ; 点検操作中
      AND     M505  ; HMI_X軸ジョグ逆転
      LD      M35  ; 地上側から_手動操作中
      AND     M525  ; 地上→手動_X軸ジョグ逆転
      ORB
      ANB
      AND     M418  ; X軸 逆回転可
      OUT     M265  ; X軸_逆回転ジョグ
      MPP
      LD      M30  ; 点検操作中
      OR      M35  ; 地上側から_手動操作中
      ANB
      LD      M264  ; X軸_正回転ジョグ
      OR      M265  ; X軸_逆回転ジョグ
      ANB
      MOV     K100 D135
      OUT     M101  ; X軸_Enable応用停止補助 2
      MOV     D5003 D131
      MOV     K50 D132
      MOV     K50 D133
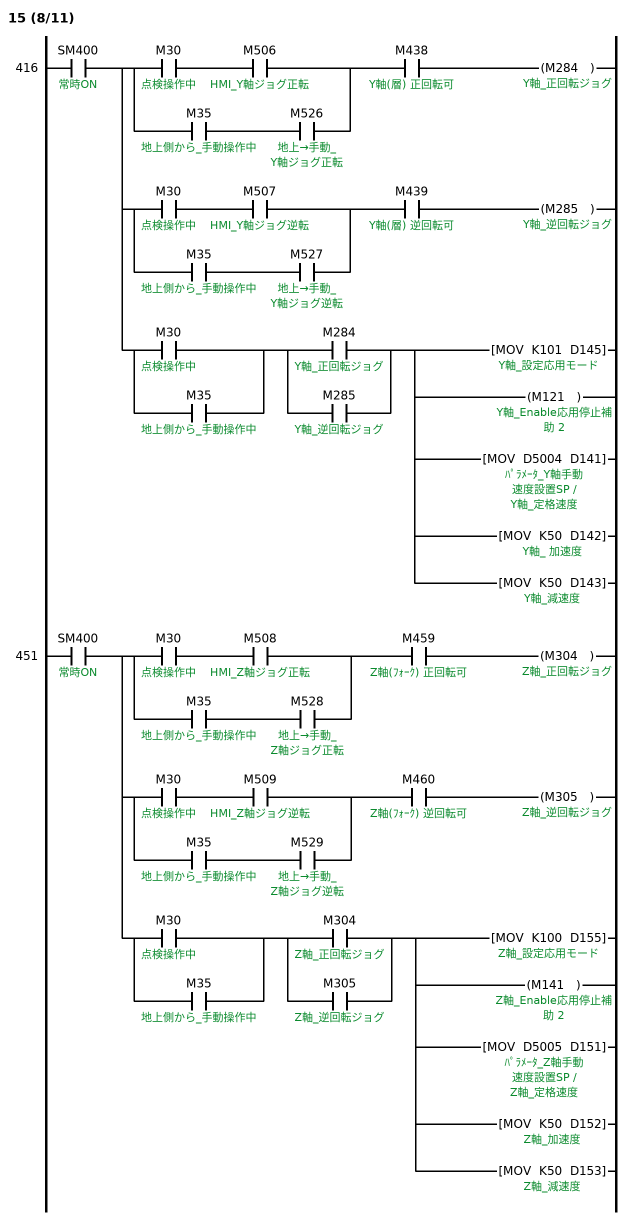
416   LD      SM400  ; 常時ON
      MPS
      LD      M30  ; 点検操作中
      AND     M506  ; HMI_Y軸ジョグ正転
      LD      M35  ; 地上側から_手動操作中
      AND     M526  ; 地上→手動_Y軸ジョグ正転
      ORB
      ANB
      AND     M438  ; Y軸(層) 正回転可
      OUT     M284  ; Y軸_正回転ジョグ
      MRD
      LD      M30  ; 点検操作中
      AND     M507  ; HMI_Y軸ジョグ逆転
      LD      M35  ; 地上側から_手動操作中
      AND     M527  ; 地上→手動_Y軸ジョグ逆転
      ORB
      ANB
      AND     M439  ; Y軸(層) 逆回転可
      OUT     M285  ; Y軸_逆回転ジョグ
      MPP
      LD      M30  ; 点検操作中
      OR      M35  ; 地上側から_手動操作中
      ANB
      LD      M284  ; Y軸_正回転ジョグ
      OR      M285  ; Y軸_逆回転ジョグ
      ANB
      MOV     K101 D145
      OUT     M121  ; Y軸_Enable応用停止補助 2
      MOV     D5004 D141
      MOV     K50 D142
      MOV     K50 D143
451   LD      SM400  ; 常時ON
      MPS
      LD      M30  ; 点検操作中
      AND     M508  ; HMI_Z軸ジョグ正転
      LD      M35  ; 地上側から_手動操作中
      AND     M528  ; 地上→手動_Z軸ジョグ正転
      ORB
      ANB
      AND     M459  ; Z軸(ﾌｫｰｸ) 正回転可
      OUT     M304  ; Z軸_正回転ジョグ
      MRD
      LD      M30  ; 点検操作中
      AND     M509  ; HMI_Z軸ジョグ逆転
      LD      M35  ; 地上側から_手動操作中
      AND     M529  ; 地上→手動_Z軸ジョグ逆転
      ORB
      ANB
      AND     M460  ; Z軸(ﾌｫｰｸ) 逆回転可
      OUT     M305  ; Z軸_逆回転ジョグ
      MPP
      LD      M30  ; 点検操作中
      OR      M35  ; 地上側から_手動操作中
      ANB
      LD      M304  ; Z軸_正回転ジョグ
      OR      M305  ; Z軸_逆回転ジョグ
      ANB
      MOV     K100 D155
      OUT     M141  ; Z軸_Enable応用停止補助 2
      MOV     D5005 D151
      MOV     K50 D152
      MOV     K50 D153
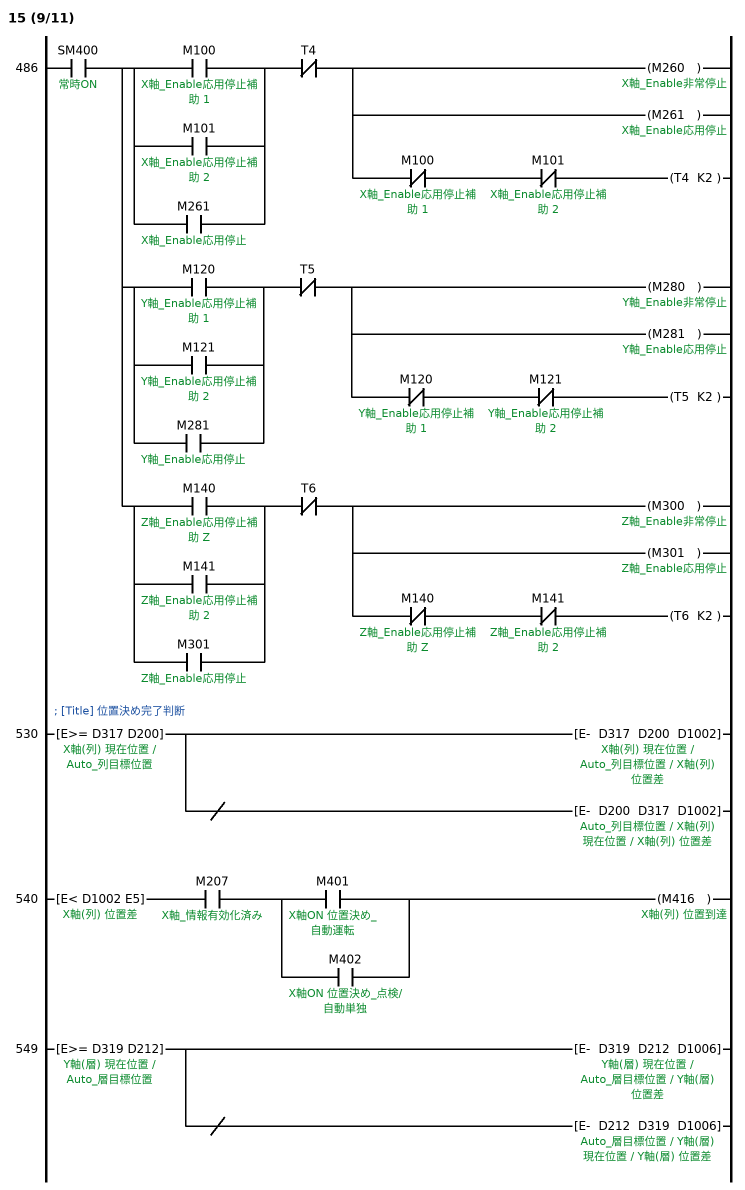
486   LD      SM400  ; 常時ON
      MPS
      LD      M100  ; X軸_Enable応用停止補助 1
      OR      M101  ; X軸_Enable応用停止補助 2
      OR      M261  ; X軸_Enable応用停止
      ANB
      ANI     T4
      OUT     M260  ; X軸_Enable非常停止
      OUT     M261  ; X軸_Enable応用停止
      ANI     M100  ; X軸_Enable応用停止補助 1
      ANI     M101  ; X軸_Enable応用停止補助 2
      OUT     T4 K2
      MRD
      LD      M120  ; Y軸_Enable応用停止補助 1
      OR      M121  ; Y軸_Enable応用停止補助 2
      OR      M281  ; Y軸_Enable応用停止
      ANB
      ANI     T5
      OUT     M280  ; Y軸_Enable非常停止
      OUT     M281  ; Y軸_Enable応用停止
      ANI     M120  ; Y軸_Enable応用停止補助 1
      ANI     M121  ; Y軸_Enable応用停止補助 2
      OUT     T5 K2
      MPP
      LD      M140  ; Z軸_Enable応用停止補助 Z
      OR      M141  ; Z軸_Enable応用停止補助 2
      OR      M301  ; Z軸_Enable応用停止
      ANB
      ANI     T6
      OUT     M300  ; Z軸_Enable非常停止
      OUT     M301  ; Z軸_Enable応用停止
      ANI     M140  ; Z軸_Enable応用停止補助 Z
      ANI     M141  ; Z軸_Enable応用停止補助 2
      OUT     T6 K2
; [Title] 位置決め完了判断
530   LDE>=   D317 D200  ; X軸(列) 現在位置 / Auto_列目標位置
      E-      D317 D200 D1002  ; X軸(列) 位置差
      INV
      E-      D200 D317 D1002
540   LDE<    D1002 E5  ; X軸(列) 位置差
      AND     M207  ; X軸_情報有効化済み
      LD      M401  ; X軸ON 位置決め_自動運転
      OR      M402  ; X軸ON 位置決め_点検/自動単独
      ANB
      OUT     M416  ; X軸(列) 位置到達
549   LDE>=   D319 D212  ; Y軸(層) 現在位置 / Auto_層目標位置
      E-      D319 D212 D1006  ; Y軸(層) 位置差
      INV
      E-      D212 D319 D1006
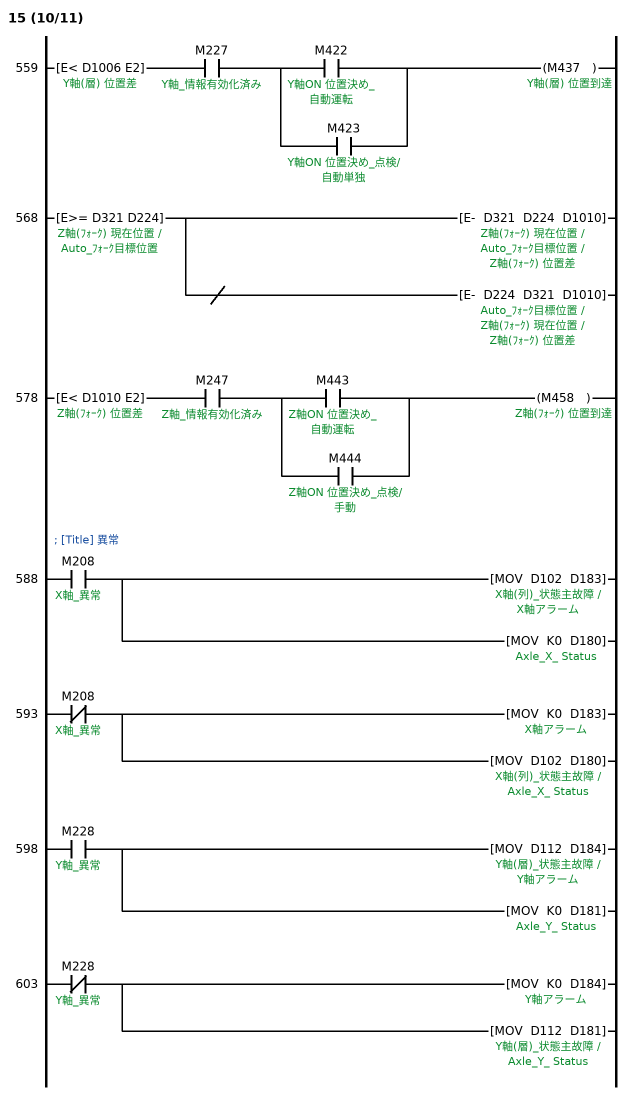
559   LDE<    D1006 E2  ; Y軸(層) 位置差
      AND     M227  ; Y軸_情報有効化済み
      LD      M422  ; Y軸ON 位置決め_自動運転
      OR      M423  ; Y軸ON 位置決め_点検/自動単独
      ANB
      OUT     M437  ; Y軸(層) 位置到達
568   LDE>=   D321 D224  ; Z軸(ﾌｫｰｸ) 現在位置 / Auto_ﾌｫｰｸ目標位置
      E-      D321 D224 D1010  ; Z軸(ﾌｫｰｸ) 位置差
      INV
      E-      D224 D321 D1010
578   LDE<    D1010 E2  ; Z軸(ﾌｫｰｸ) 位置差
      AND     M247  ; Z軸_情報有効化済み
      LD      M443  ; Z軸ON 位置決め_自動運転
      OR      M444  ; Z軸ON 位置決め_点検/手動
      ANB
      OUT     M458  ; Z軸(ﾌｫｰｸ) 位置到達
; [Title] 異常
588   LD      M208  ; X軸_異常
      MOV     D102 D183  ; X軸(列)_状態主故障 / X軸アラーム
      MOV     K0 D180  ; Axle_X_ Status
593   LDI     M208  ; X軸_異常
      MOV     K0 D183
      MOV     D102 D180
598   LD      M228  ; Y軸_異常
      MOV     D112 D184  ; Y軸(層)_状態主故障 / Y軸アラーム
      MOV     K0 D181  ; Axle_Y_ Status
603   LDI     M228  ; Y軸_異常
      MOV     K0 D184
      MOV     D112 D181
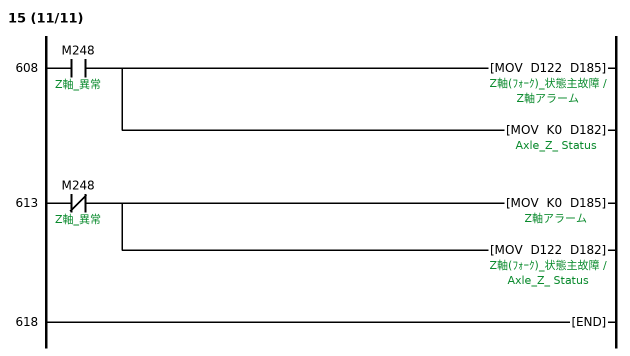
608   LD      M248  ; Z軸_異常
      MOV     D122 D185  ; Z軸(ﾌｫｰｸ)_状態主故障 / Z軸アラーム
      MOV     K0 D182  ; Axle_Z_ Status
613   LDI     M248  ; Z軸_異常
      MOV     K0 D185
      MOV     D122 D182
618   END
END_PROGRAM

PROGRAM 50  // I/O出力
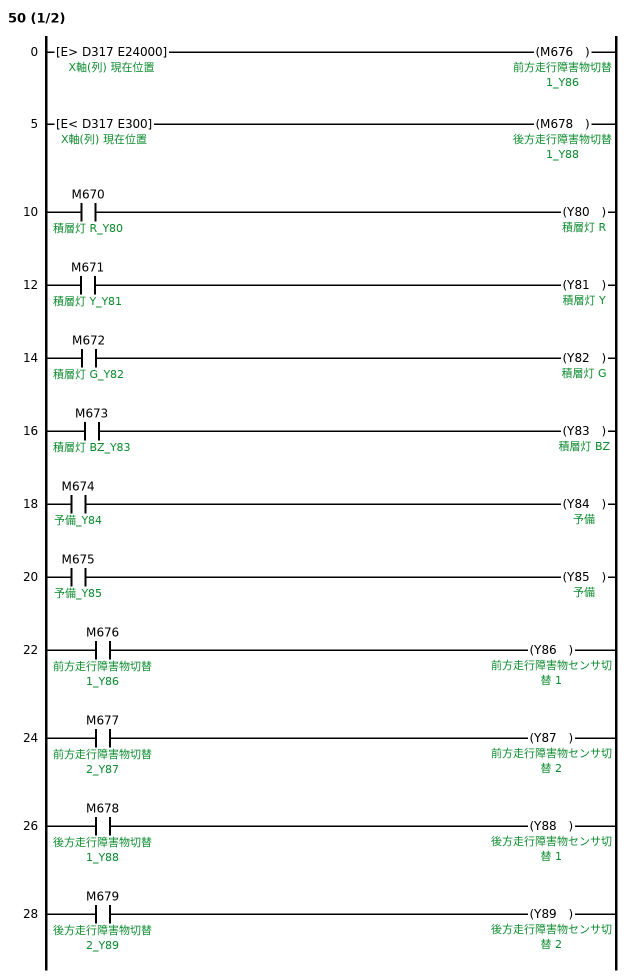
0     LDE>    D317 E24000  ; X軸(列) 現在位置
      OUT     M676  ; 前方走行障害物切替 1_Y86
5     LDE<    D317 E300  ; X軸(列) 現在位置
      OUT     M678  ; 後方走行障害物切替 1_Y88
10    LD      M670  ; 積層灯 R_Y80
      OUT     Y80  ; 積層灯 R
12    LD      M671  ; 積層灯 Y_Y81
      OUT     Y81  ; 積層灯 Y
14    LD      M672  ; 積層灯 G_Y82
      OUT     Y82  ; 積層灯 G
16    LD      M673  ; 積層灯 BZ_Y83
      OUT     Y83  ; 積層灯 BZ
18    LD      M674  ; 予備_Y84
      OUT     Y84  ; 予備
20    LD      M675  ; 予備_Y85
      OUT     Y85  ; 予備
22    LD      M676  ; 前方走行障害物切替 1_Y86
      OUT     Y86  ; 前方走行障害物センサ切替 1
24    LD      M677  ; 前方走行障害物切替 2_Y87
      OUT     Y87  ; 前方走行障害物センサ切替 2
26    LD      M678  ; 後方走行障害物切替 1_Y88
      OUT     Y88  ; 後方走行障害物センサ切替 1
28    LD      M679  ; 後方走行障害物切替 2_Y89
      OUT     Y89  ; 後方走行障害物センサ切替 2
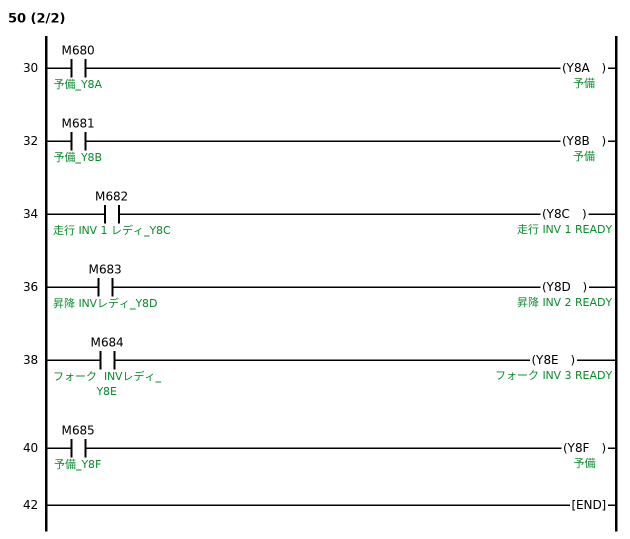
30    LD      M680  ; 予備_Y8A
      OUT     Y8A  ; 予備
32    LD      M681  ; 予備_Y8B
      OUT     Y8B  ; 予備
34    LD      M682  ; 走行 INV 1 レディ_Y8C
      OUT     Y8C  ; 走行 INV 1 READY
36    LD      M683  ; 昇降 INVレディ_Y8D
      OUT     Y8D  ; 昇降 INV 2 READY
38    LD      M684  ; フォーク  INVレディ_Y8E
      OUT     Y8E  ; フォーク INV 3 READY
40    LD      M685  ; 予備_Y8F
      OUT     Y8F  ; 予備
42    END
END_PROGRAM

PROGRAM 21  // 安全機器有効無効
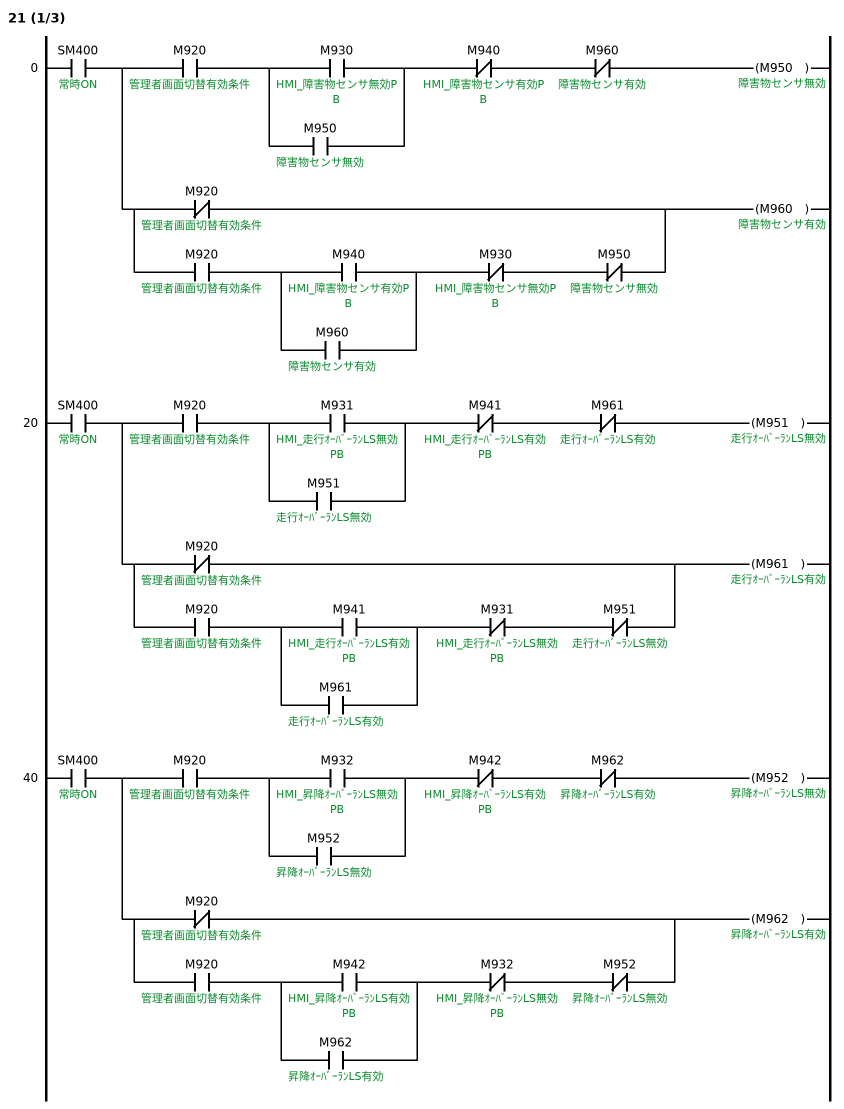
0     LD      SM400  ; 常時ON
      MPS
      AND     M920  ; 管理者画面切替有効条件
      LD      M930  ; HMI_障害物センサ無効PB
      OR      M950  ; 障害物センサ無効
      ANB
      ANI     M940  ; HMI_障害物センサ有効PB
      ANI     M960  ; 障害物センサ有効
      OUT     M950  ; 障害物センサ無効
      MPP
      LDI     M920  ; 管理者画面切替有効条件
      LD      M920  ; 管理者画面切替有効条件
      LD      M940  ; HMI_障害物センサ有効PB
      OR      M960  ; 障害物センサ有効
      ANB
      ANI     M930  ; HMI_障害物センサ無効PB
      ANI     M950  ; 障害物センサ無効
      ORB
      ANB
      OUT     M960  ; 障害物センサ有効
20    LD      SM400  ; 常時ON
      MPS
      AND     M920  ; 管理者画面切替有効条件
      LD      M931  ; HMI_走行ｵｰﾊﾞｰﾗﾝLS無効PB
      OR      M951  ; 走行ｵｰﾊﾞｰﾗﾝLS無効
      ANB
      ANI     M941  ; HMI_走行ｵｰﾊﾞｰﾗﾝLS有効PB
      ANI     M961  ; 走行ｵｰﾊﾞｰﾗﾝLS有効
      OUT     M951  ; 走行ｵｰﾊﾞｰﾗﾝLS無効
      MPP
      LDI     M920  ; 管理者画面切替有効条件
      LD      M920  ; 管理者画面切替有効条件
      LD      M941  ; HMI_走行ｵｰﾊﾞｰﾗﾝLS有効PB
      OR      M961  ; 走行ｵｰﾊﾞｰﾗﾝLS有効
      ANB
      ANI     M931  ; HMI_走行ｵｰﾊﾞｰﾗﾝLS無効PB
      ANI     M951  ; 走行ｵｰﾊﾞｰﾗﾝLS無効
      ORB
      ANB
      OUT     M961  ; 走行ｵｰﾊﾞｰﾗﾝLS有効
40    LD      SM400  ; 常時ON
      MPS
      AND     M920  ; 管理者画面切替有効条件
      LD      M932  ; HMI_昇降ｵｰﾊﾞｰﾗﾝLS無効PB
      OR      M952  ; 昇降ｵｰﾊﾞｰﾗﾝLS無効
      ANB
      ANI     M942  ; HMI_昇降ｵｰﾊﾞｰﾗﾝLS有効PB
      ANI     M962  ; 昇降ｵｰﾊﾞｰﾗﾝLS有効
      OUT     M952  ; 昇降ｵｰﾊﾞｰﾗﾝLS無効
      MPP
      LDI     M920  ; 管理者画面切替有効条件
      LD      M920  ; 管理者画面切替有効条件
      LD      M942  ; HMI_昇降ｵｰﾊﾞｰﾗﾝLS有効PB
      OR      M962  ; 昇降ｵｰﾊﾞｰﾗﾝLS有効
      ANB
      ANI     M932  ; HMI_昇降ｵｰﾊﾞｰﾗﾝLS無効PB
      ANI     M952  ; 昇降ｵｰﾊﾞｰﾗﾝLS無効
      ORB
      ANB
      OUT     M962  ; 昇降ｵｰﾊﾞｰﾗﾝLS有効
